// TIA Portal V17 export
// export: Created 2022-03-12T16:05:16.204313Z, ExportSetting WithDefaults, DisplayName Totally Integrated Automation Portal, DisplayVersion V17, DisplayName TIA Portal Openness, DisplayVersion V17, DisplayName TIA Portal Version Control Interface, DisplayVersion V17, DisplayName STEP 7 Professional, DisplayVersion V17, DisplayName STEP 7 Safety, DisplayVersion V17, DisplayName WinCC Advanced / Unified PC, DisplayVersion V17
DATA_BLOCK "UN"   // DB31629
TITLE = UN
{ S7_Optimized_Access := 'TRUE' }
AUTHOR : tech.team.motioncontrol@siemens.com
FAMILY : CPG
VERSION : 1.0
// Support: tech.team.motioncontrol@siemens.com
// Fax: +49 (0) 9131/98-1297
// stored: AutoNumber true, DBAccessibleFromOPCUA true, DBAccessibleFromWebserver true, IsOnlyStoredInLoadMemory false, IsRetainMemResEnabled false, IsWriteProtectedInAS false, MemoryReserve 100
   VAR
      PackML_Sts { ExternalWritable := 'False'; S7_SetPoint := 'True'} : "CPG_typePackML_ModuleSts";   // PackML Module Status - UN Status
      PackML_Sts_Alarm { ExternalWritable := 'False'; S7_SetPoint := 'True'} : "CPG_typePackML_ModuleSts";   // PackML Module Status - UN alarm status
      Alarm { ExternalAccessible := 'False'; ExternalVisible := 'False'; ExternalWritable := 'False'; S7_SetPoint := 'True'} : "CPG_typeEventStatus";   // Alarm Event Status - UN Status
      Warning { ExternalAccessible := 'False'; ExternalVisible := 'False'; ExternalWritable := 'False'; S7_SetPoint := 'True'} : "CPG_typeEventStatus";   // Warning Event Status - UN Status
      Status { ExternalAccessible := 'False'; ExternalVisible := 'False'; ExternalWritable := 'False'; S7_SetPoint := 'True'} : "CPG_typeEventStatus";   // Event Status - UN Status
   END_VAR
BEGIN
END_DATA_BLOCK
